TYPE DUT_HMI_11_MANUALS :
STRUCT
	PS : ARRAY[0..CNC.NUM_MAX_MANUALS_11-1] OF BOOL;
	LS : ARRAY[0..CNC.NUM_MAX_MANUALS_11-1] OF BOOL;
END_STRUCT
END_TYPE

(* stored: Version 1.1.0.1, ProductVersion 3.1.4024.13
   DUT DUT_HMI_11_MANUALS: Id {41e42190-e20a-41dc-a6d8-323390bcef76} *)
